FUNCTION_BLOCK E_CYCLE (* Periodic (cyclic) Generation of an Event (synthetic test fixture 26.0.0.7) *)
  (* Standard: 61499-1 *)
  PACKAGE IEC61499.Standard;
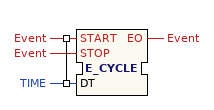
  EVENT_INPUT
    START WITH DT;
    STOP;
  END_EVENT
  EVENT_OUTPUT
    EO;
  END_EVENT
  VAR_INPUT
    DT : TIME; (* Period between events *)
  END_VAR
END_FUNCTION_BLOCK
